PROGRAM MAIN
VAR
	fbO5D100 : Identical_Library.FB_O5D100;
END_VAR

fbO5D100();

END_PROGRAM

(* stored: Version 1.1.0.1, ProductVersion 3.1.4024.12
   POU MAIN: Id {802e6176-3be3-4153-b01c-d723f6ad006d}, SpecialFunc None *)
